{attribute wpf [Container(Layout.Stack)]}
FUNCTION_BLOCK Station001_Components EXTENDS TcoCore.TcoObject
VAR	
//	_horizontalAxis : DriveSim(THIS^);
	{attribute addProperty Name "Horizontal axis"}
	_horizontalNcAxis : TcoDrivesBeckhoff.TcoDriveSimple(THIS^); 
	{attribute addProperty Name "Vertical piston"}
	_verticalPiston : TcoPneumatics.TcoCylinder(THIS^);
	{attribute addProperty Name "Gripper piston"}
	_gripperPiston : TcoPneumatics.TcoCylinder(THIS^);
END_VAR
(* Simulation variables *)
VAR
	_counterSimVerticalPiston : ULINT;
	_counterSimGripperPiston : ULINT;
	_simulationCycleVerticalPiston : BOOL;	
	_simulationCycleGripperPiston : BOOL;	
	_verticalPosition : INT;
	_gripperPosition : INT;
	_dimXsim : RealValueSimulation;
	_dimYsim : RealValueSimulation;
	_dimZsim : RealValueSimulation;
	_dimX : REAL;
	_dimY : REAL;
	_dimZ : REAL;
END_VAR
VAR CONSTANT
	_verticalPistonStroke : INT := 150;
	_gripperPistonStroke : INT := 50;
END_VAR

Simulation();

_verticalPiston(inoAtHomePos := IO.iA1[0],
    inoAtWorkPos := IO.iA1[1],
    inoToHomePos := IO.qA1[0],
    inoToWorkPos := IO.qA1[1]);

_gripperPiston(inoAtHomePos := IO.iA1[2],
    inoAtWorkPos := IO.iA1[3],
    inoToHomePos := IO.qA1[2],
    inoToWorkPos := IO.qA1[3]);

//_horizontalAxis();
_horizontalNcAxis(inEnable := TRUE,
    inEnablePositive := TRUE,
    inEnableNegative := TRUE,
    inCalibrationCam := FALSE,
    inoAxisRef := IO.Axis1);

PROPERTY Gripper :  REFERENCE TO TcoPneumatics.TcoCylinder
GET
Gripper REF= _gripperPiston;
END_GET
END_PROPERTY

PROPERTY HorizontalNcAxis : TcoDrivesBeckhoff.ITcoDriveSimple
GET
HorizontalNcAxis := _horizontalNcAxis;
END_GET
END_PROPERTY

METHOD Service : BOOL
VAR_INPUT
END_VAR
//_horizontalAxis.Service();
_horizontalNcAxis.Service();
_verticalPiston.Service();
_gripperPiston.Service();
END_METHOD

METHOD Simulation
VAR_INPUT
END_VAR
IF (_verticalPiston.MoveHomeTask.Busy OR _verticalPiston.MoveWorkTask.Busy) THEN
    _counterSimVerticalPiston := _counterSimVerticalPiston + 1;
    _simulationCycleVerticalPiston := (_counterSimVerticalPiston MOD _verticalPistonStroke) = 0;
END_IF;

IF (Gripper.MoveHomeTask.Busy OR Gripper.MoveWorkTask.Busy) THEN
    _counterSimGripperPiston := _counterSimVerticalPiston + 1;
    _simulationCycleGripperPiston := (_counterSimVerticalPiston MOD _gripperPistonStroke) = 0;
END_IF;

IF (IO.qA1[0] AND _simulationCycleVerticalPiston) THEN
    IO.iA1[0] := TRUE;
    IO.iA1[1] := FALSE;
    _verticalPosition := 0;
END_IF

IF (IO.qA1[1] AND _simulationCycleVerticalPiston) THEN
    IO.iA1[1] := TRUE;
    IO.iA1[0] := FALSE;
    _verticalPosition := _verticalPistonStroke;
END_IF

IF (IO.qA1[0] AND NOT IO.iA1[0]) THEN
    _verticalPosition := (_verticalPosition - 1);
END_IF;

IF (IO.qA1[1] AND NOT IO.iA1[1]) THEN
    _verticalPosition := (_verticalPosition + 1);
END_IF;

IF (IO.qA1[2] AND _simulationCycleVerticalPiston) THEN
    IO.iA1[2] := TRUE;
    IO.iA1[3] := FALSE;
    _gripperPosition := 0;
END_IF

IF (IO.qA1[3] AND _simulationCycleVerticalPiston) THEN
    IO.iA1[3] := TRUE;
    IO.iA1[2] := FALSE;
    _gripperPosition := _gripperPistonStroke;
END_IF

IF (IO.qA1[2] AND NOT IO.iA1[2]) THEN
    _gripperPosition := (_gripperPosition - 1);
END_IF;

IF (IO.qA1[3] AND NOT IO.iA1[3]) THEN
    _gripperPosition := (_gripperPosition + 1);
END_IF

_dimXsim.Dc := 3;
_dimYsim.Dc := 3;
_dimZsim.Dc := 3;
_dimXsim.P1 := 0.74;
_dimYsim.P1 := 0.74;
_dimZsim.P1 := 0.74;
_dimXsim.P2 := 1.1;
_dimYsim.P2 := 1.1;
_dimZsim.P2 := 1.1;
END_METHOD

PROPERTY VerticalAxis : REFERENCE TO TcoPneumatics.TcoCylinder
GET
VerticalAxis REF= _verticalPiston;
END_GET
END_PROPERTY

END_FUNCTION_BLOCK

(* stored: Version 1.1.0.1, ProductVersion 3.1.4024.9
   POU Station001_Components: Id {e806c847-ecc4-43b0-a026-69e0b11f80ef}, SpecialFunc None
   Property Gripper: Id {45058c8f-3b79-49b6-8729-6389402fa4b0}
   Get Get: Id {d387ff5f-f5d6-44a8-b450-cb493513cbfe}
   Property HorizontalNcAxis: Id {50ed9664-d5a7-4e96-a637-5203276f92d3}
   Get Get: Id {a7390b8e-0434-4b57-9dfc-bdeb3f9087e0}
   Method Service: Id {98457207-8a91-45fe-bd57-5bb0d15033a9}
   Method Simulation: Id {2b05f176-ee43-4d85-a715-7bea1c119c16}
   Property VerticalAxis: Id {95519e2e-c8d9-4542-adf0-78464b1acba5}
   Get Get: Id {2a859788-f8eb-4b2b-8a8a-19eb876b8488} *)
